PROGRAM PRG_MFuncControl
VAR
	bActivateTool		: BOOL;
END_VAR

IF NCI.bMFunc[5] THEN
	bActivateTool			:= TRUE;
	NCI.bQuitMFunc[11]		:= TRUE;
END_IF


IF NCI.bMFunc[12] THEN
	bActivateTool			:= FALSE;
	NCI.bQuitMFunc[12]		:= TRUE;
END_IF

END_PROGRAM

(* stored: Version 1.1.0.1, ProductVersion 3.1.4024.10
   POU PRG_MFuncControl: Id {19677d06-9e27-4323-bf51-bb01aefc8330}, SpecialFunc None *)
